Staubli VAL3: onExit.pgx

program onExit(bool& x_bSave[] (dimensions=1))
  local string l_sMessage
  local bool l_bYes
  local bool l_bCancel
  local string l_sButton[2]
begin
  // saveIt
  if x_bSave
    call language:message(l_sMessage,-1)
    call language:getYesNo(l_sButton)
    // ask the yes_no question
    call use:yes_no_cancel(l_sMessage,l_sButton,l_bYes,l_bCancel)
    if l_bYes
      call saveIt(x_bSave)
    endIf
    // look for the cancel button
    bExit=!l_bCancel
  else
    // exit frome the page
    bExit=true
  endIf
  // send Back
  if size(sItems)>1
    sItems[1]=toString("",nIndexItem)
  endIf
  // null key
  call use:nullKey(nKey)
  // reset the show status
  bShowStatus=false
  // resetMotion
  if !cycleStatus:bCycle
    resetMotion()
  endIf
end
